TYPE IonizerConfigs :
STRUCT
	SJH108IonizerConfig : SJH108IonizerConfig;
END_STRUCT
END_TYPE

(* stored: Version 1.1.0.1, ProductVersion 3.1.4024.12
   DUT IonizerConfigs: Id {95492f59-ea68-4416-9597-fc69d0b77b59} *)
